// TIA Portal V17 export
// export: Created 2025-06-26T07:49:14.0746139Z, ExportSetting WithDefaults, DisplayName Totally Integrated Automation Portal, DisplayVersion V17 Update 8, DisplayName TIA Portal Openness, DisplayVersion V17 Update 8, DisplayName TIA Portal Version Control Interface, DisplayVersion V17, DisplayName STEP 7 Professional, DisplayVersion V17 Update 8, DisplayName STEP 7 Safety, DisplayVersion V17 Update 6, DisplayName WinCC Advanced, DisplayVersion V17 Update 8
DATA_BLOCK "CAN-Communication_DB"   // DB14
VERSION : 0.1
// stored: AutoNumber false, DBAccessibleFromOPCUA true, InstanceOfName CAN-Communication, InstanceOfType FB
"CAN-Communication"
   // VAR_IN_OUT
   //    "CAN-IDs_ToSend" : Array[0..74] of Int;
   // END_VAR
   // VAR
   //    SendBusy : Bool;
   //    UseFixedPoint : Bool;
   //    Memory : DInt;
   //    CycleCheck : Bool;
   //    TESTUINT_CTRL { ExternalAccessible := 'False'; ExternalVisible := 'False'; ExternalWritable := 'False'} : UInt;
   //    TESTUINT_SEND : UInt;
   //    TESTUINT_RCV : UInt;
   //    TOF_SendError { S7_SetPoint := 'True'} : TOF_TIME;
   //    CountSendAll : UDInt;
   //    ScaleFactor : Real;
   // END_VAR
BEGIN
END_DATA_BLOCK
